{attribute 'qualified_only'}
{attribute 'strict'}
TYPE E_DisplayFormat :
(
    Decimal := 0,
    Binary  := 1,
    Hex     := 2
);
END_TYPE

(* stored: Version 1.1.0.1
   EnumerationTextList E_DisplayFormat: Id {4f197284-34e6-0a19-0ed9-8abc72ed02a2} *)
